{attribute 'qualified_only'}
VAR_GLOBAL
	TST_OUT AT%Q*	: BYTE;
END_VAR

(* stored: Version 1.1.0.1, ProductVersion 3.1.4024.12
   GVL GVL_TEST: Id {2f563851-8a7d-4ba9-bae9-f568d15b16c6} *)
